// TIA Portal V19 export
TYPE "lexchangetray_typeUnEmn_deliver_interface"
// Type: lexchangetray_typeUnEmn_toHandlingXyzDeliver
// Type: lexchangetray_typeUnEmn_toConstraintWorkstationDeliver
// Type: lexchangetray_typeUnEmn_toRollerDeliver
// Type: Bool
// stored: Access Published
   STRUCT
      init : Bool;
      roller : "lexchangetray_typeUnEmn_toRollerDeliver";
      constraintWorkstation { S7_SetPoint := 'True'} : "lexchangetray_typeUnEmn_toConstraintWorkstationDeliver";
      handlingXyz { S7_SetPoint := 'True'} : "lexchangetray_typeUnEmn_toHandlingXyzDeliver";
   END_STRUCT;
END_TYPE
